Staubli VAL3: SimuMain.pgx

public program SimuMain(string x_sPath)
  local num l_nKey
begin
  //
  bExit=false
  bUserRefresh=bListRefresh=true
  sPath=x_sPath
  do
    call Refresh2()
    call RefreshList()
    call user:setList("路径",sList,bUserRefresh,bListRefresh,nSelected,sItem,l_nKey)
    bUserRefresh=false
    bListRefresh=false
    call MainKey(l_nKey)
    delay(0)
  until bExit
  bUserRefresh=bListRefresh=true
  bExit=false
end
